{attribute 'linkalways'} 
{attribute 'no_explicit_call' := 'This FB is a CLASS and must be accessed using methods or properties'}
{attribute 'enable_dynamic_creation'}
FUNCTION_BLOCK Session EXTENDS Disposable IMPLEMENTS I_Session
VAR
	_id : T_MAXSTRING;
	_lastAccessedTimestamp : SystemTimestamp;
	sessionStorage : Dictionary;
END_VAR

METHOD PUBLIC AddOrUpdateStorage
VAR_INPUT
	StorageId : T_MAXSTRING;
	Source : I_SessionData;
END_VAR
sessionStorage.AddOrUpdate(StorageId, Source);
END_METHOD

METHOD PUBLIC DisposeAllDataFromStorage
VAR_INPUT
END_VAR
VAR
	enumerator : I_ForwardEnumerator;
	sessionData : I_SessionData;
END_VAR
enumerator := sessionStorage.GetEnumerator();

WHILE enumerator.MoveNext() DO
	IF enumerator.TryGet(sessionData) THEN
		sessionData.Dispose();
	END_IF
END_WHILE

enumerator.Dispose();
sessionStorage.Clear();
END_METHOD

METHOD PUBLIC DisposeDataFromStorage
VAR_INPUT
	StorageId : T_MAXSTRING;
END_VAR
VAR
	sessionData : I_SessionData;
END_VAR
IF NOT sessionStorage.TryGetValue(StorageId,sessionData) THEN
	RETURN;
END_IF

sessionData.Dispose();
sessionStorage.Remove(StorageId);
END_METHOD

METHOD FB_exit : BOOL
VAR_INPUT
	bInCopyCode : BOOL; // if TRUE, the exit method is called for exiting an instance that is copied afterwards (online change).
END_VAR
IF bInCopyCode THEN
	RETURN;
END_IF

DisposeAllDataFromStorage();
END_METHOD

METHOD FB_init : BOOL
VAR_INPUT
	bInitRetains : BOOL; // if TRUE, the retain variables are initialized (warm start / cold start)
	bInCopyCode : BOOL;  // if TRUE, the instance afterwards gets moved into the copy code (online change)
	SessionId : T_MAXSTRING;
END_VAR
_id := SessionId;
END_METHOD

PROPERTY PUBLIC Id : T_MAXSTRING
GET
Id := _id;
END_GET
END_PROPERTY

PROPERTY PUBLIC LastAccessedTimestamp : I_TimeStamp
GET
LastAccessedTimestamp := _lastAccessedTimestamp;
END_GET
END_PROPERTY

METHOD PUBLIC Refresh
VAR_INPUT
END_VAR
_lastAccessedTimestamp.SetNow();
END_METHOD

METHOD PUBLIC TryGetDataFromStorage : BOOL
VAR_INPUT
	StorageId : T_MAXSTRING;
	Destination : REFERENCE TO I_SessionData;
END_VAR
TryGetDataFromStorage := sessionStorage.TryGetValue(StorageId, Destination);
END_METHOD

END_FUNCTION_BLOCK

(* stored: Version 1.1.0.1, ProductVersion 3.1.4024.12
   POU Session: Id {dc893d80-001c-0432-282c-2031ac3cf2c1}, SpecialFunc None
   Folder Constructor: Id {c2a1fc72-b779-0673-3e14-f35c61ae51d0}
   Folder Destructor: Id {ec7f9341-6488-0e65-1036-613ebb9bf0ac}
   Method AddOrUpdateStorage: Id {afc67cb0-d360-0d99-0988-4c146c0ce805}
   Method DisposeAllDataFromStorage: Id {8a6c5779-1368-0954-126f-e291e6b2ff7a}
   Method DisposeDataFromStorage: Id {1d4a66d1-cd79-0563-0a05-eb32943e2977}
   Method FB_exit: Id {6dc69cf5-f7ae-0e42-2cba-1c6d0aa20592}
   Method FB_init: Id {7dca8727-0db7-0ed6-0e80-88e544397ad3}
   Property Id: Id {dcfb7953-5fef-015f-3827-7ebdd268e7b5}
   Get Get: Id {ee886ace-15dc-06ad-31d8-c447d377f50b}
   Property LastAccessedTimestamp: Id {6ae8e0fa-f398-044b-0522-fede2eababc1}
   Get Get: Id {7decb6cf-55cb-05a3-186d-cb1a653febd6}
   Method Refresh: Id {0674f60f-af84-0c03-061a-f0b6dc67598c}
   Method TryGetDataFromStorage: Id {43ce750e-acb3-0b7f-2b91-2ab3115909d2} *)
